PROGRAM MAIN
VAR
END_VAR

END_PROGRAM

(* stored: Version 1.1.0.1
   POU MAIN: Id {30d36252-c1e0-42c8-bfb3-99d45c6bd9d1} *)
